// TIA Portal V20 export
TYPE "LKinCtrl_typeConveyorParameter"
   STRUCT
      conveyorParaNo : DInt := 0;   // selection of conveyor parameter set from configuration structure
   END_STRUCT;
END_TYPE
